{attribute 'qualified_only'}
VAR_GLOBAL
	dummyBool	: BOOL;
END_VAR

(* stored: Version 1.1.0.1, ProductVersion 3.1.4024.12
   GVL GVL: Id {851ae7e7-1309-403f-8074-2500cd8a4e00} *)
